// SIMATIC S7-200 project (STEP 7-Micro/WIN), CPU 224 REL 01.22

ORGANIZATION_BLOCK 主程序:OB1
TITLE=程序注释
BEGIN
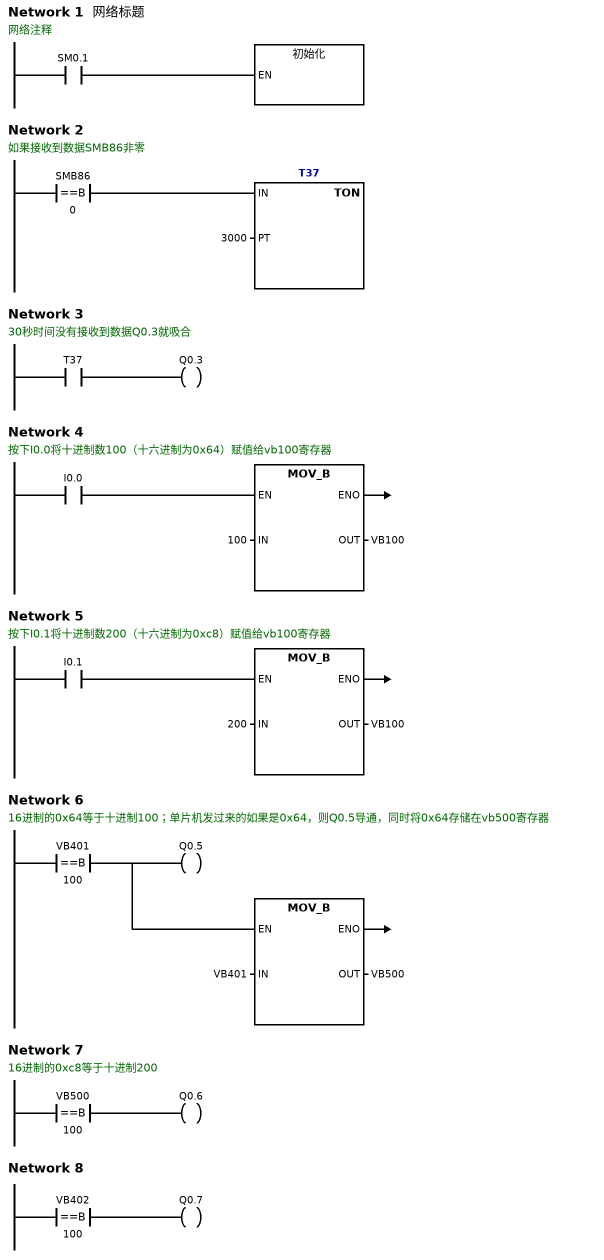
Network 1 // 网络标题
// 网络注释
LD     SM0.1
CALL   初始化:SBR0
Network 2
// 如果接收到数据SMB86非零
LDB=   SMB86, 0
TON    T37, 3000
Network 3
// 30秒时间没有接收到数据Q0.3就吸合
LD     T37
=      Q0.3
Network 4
// 按下I0.0将十进制数100（十六进制为0x64）赋值给vb100寄存器
LD     I0.0
MOVB   100, VB100
Network 5
// 按下I0.1将十进制数200（十六进制为0xc8）赋值给vb100寄存器
LD     I0.1
MOVB   200, VB100
Network 6
// 16进制的0x64等于十进制100；单片机发过来的如果是0x64，则Q0.5导通，同时将0x64存储在vb500寄存器
LDB=   VB401, 100
=      Q0.5
MOVB   VB401, VB500
Network 7
// 16进制的0xc8等于十进制200
LDB=   VB500, 100
=      Q0.6
Network 8
LDB=   VB402, 100
=      Q0.7
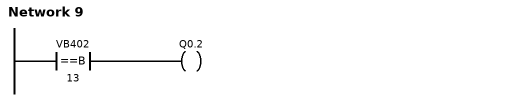
Network 9
LDB=   VB402, 13
=      Q0.2
END_ORGANIZATION_BLOCK

SUBROUTINE_BLOCK 初始化:SBR0
TITLE=子程序注释
BEGIN
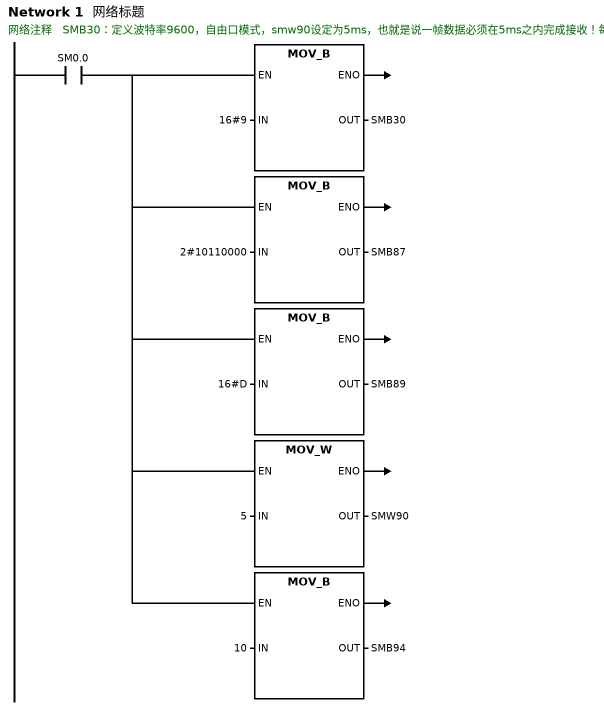
Network 1 // 网络标题
// 网络注释   SMB30：定义波特率9600，自由口模式，smw90设定为5ms，也就是说一帧数据必须在5ms之内完成接收！每次最多接收10个字节。
LD     SM0.0
MOVB   16#9, SMB30
MOVB   2#10110000, SMB87
MOVB   16#D, SMB89
MOVW   5, SMW90
MOVB   10, SMB94
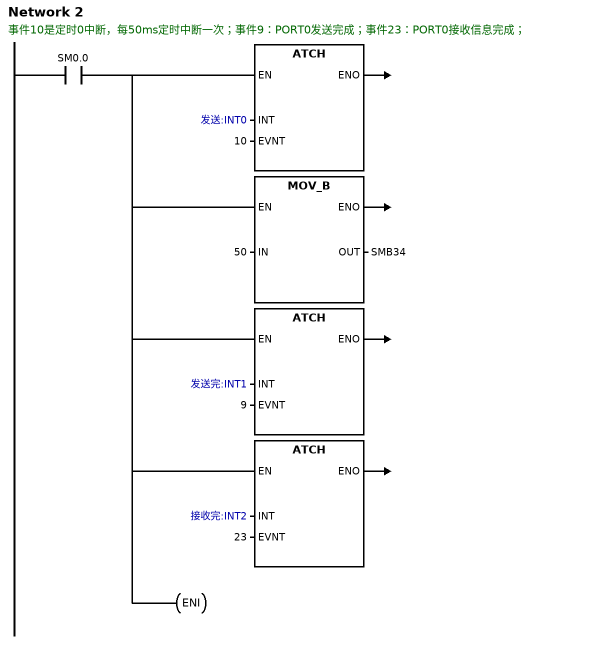
Network 2
// 事件10是定时0中断，每50ms定时中断一次；事件9：PORT0发送完成；事件23：PORT0接收信息完成；
LD     SM0.0
ATCH   发送:INT0, 10
MOVB   50, SMB34
ATCH   发送完:INT1, 9
ATCH   接收完:INT2, 23
ENI
END_SUBROUTINE_BLOCK

INTERRUPT_BLOCK 发送:INT0
TITLE=中断程序注释
BEGIN
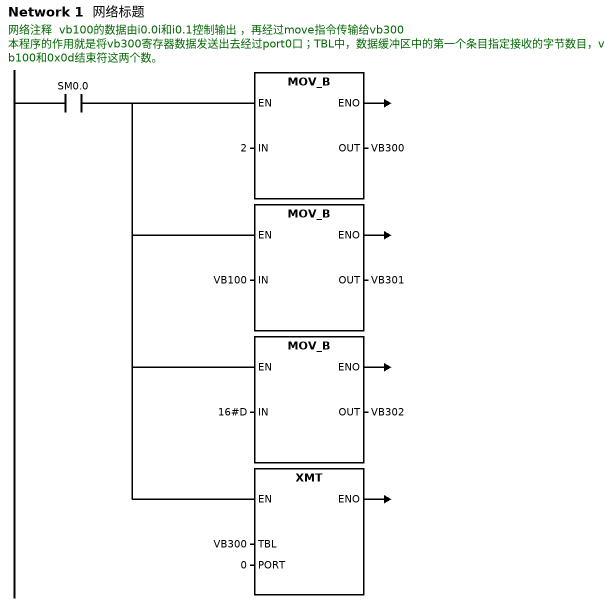
Network 1 // 网络标题
// 网络注释  vb100的数据由i0.0i和i0.1控制输出 ，再经过move指令传输给vb300   本程序的作用就是将vb300寄存器数据发送出去经过port0口；TBL中，数据缓冲区中的第一个条目指定接收的字节数目，vb300中存储的数代表要接收的数，本例中即代表要接收2个数，其中0x0d是结束符，要发送的数就是vb100和0x0d结束符这两个数。
LD     SM0.0
MOVB   2, VB300
MOVB   VB100, VB301
MOVB   16#D, VB302
XMT    VB300, 0
END_INTERRUPT_BLOCK

INTERRUPT_BLOCK 发送完:INT1
TITLE=中断程序注释
BEGIN
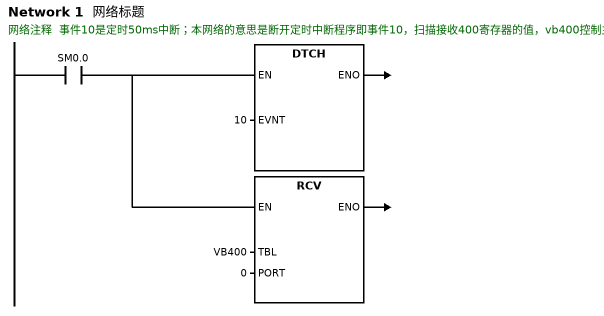
Network 1 // 网络标题
// 网络注释  事件10是定时50ms中断；本网络的意思是断开定时中断程序即事件10，扫描接收400寄存器的值，vb400控制主程序Q0.5和Q0.6；vb400字节存储的是指定接收的字节数目；vb401才是真正的接收到的数据。
LD     SM0.0
DTCH   10
RCV    VB400, 0
END_INTERRUPT_BLOCK

INTERRUPT_BLOCK 接收完:INT2
TITLE=中断程序注释
BEGIN
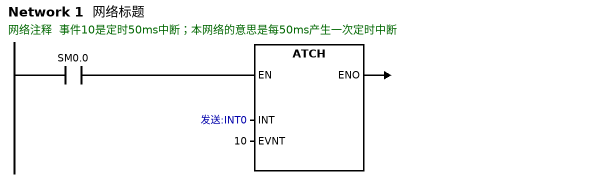
Network 1 // 网络标题
// 网络注释  事件10是定时50ms中断；本网络的意思是每50ms产生一次定时中断
LD     SM0.0
ATCH   发送:INT0, 10
END_INTERRUPT_BLOCK
